FUNCTION_BLOCK FB_Default EXTENDS FB_SeasonBase
VAR
END_VAR

METHOD  NextSeason
VAR_INST
    fbCallCtrl:     FB_InvocationControl;
END_VAR
IF fbCallCtrl.Track().bNewInvocation THEN
    Tc2_System.ADSLOGSTR(msgCtrlMask := THIS^._nLogLevel,
                         msgFmtStr := 'Current state for %s is not initialized!',
                         strArg := THIS^.sPath);
END_IF

IF THIS^.ipStateMachine <> 0 THEN
    THIS^.ipStateMachine.SetState(THIS^);
END_IF
END_METHOD

END_FUNCTION_BLOCK

(* stored: Version 1.1.0.1, ProductVersion 3.1.4024.12
   POU FB_Default: Id {95491ce9-d0ae-490b-8633-3b508fc55304}, SpecialFunc None
   Method NextSeason: Id {6eb51833-993b-4c04-8c8d-772358152a7a} *)
